(* Logix 5000 project; controller CipDriveFaultCodes vendor 1 type 14 code 156 rev 32.11; software revision 32.02 *)

TASK MainTask (continuous, watchdog 500 ms) : MainProgram

MODULES
   Local : vendor 1 type 14 code 156 (Compact 0, rev 32.11)
      Drive_1 : vendor 1 type 37 code 46 (Ethernet 192.168.1.26, rev 7.8, MotionDiagnostics RPI 1 ms)
END_MODULES

VAR_GLOBAL   (* controller tags *)
   A1_CIPAxisFaultsLSW : DINT;
   A1_CIPAxisFaultsMSW : DINT := 45;
   A1_CIPAxisFaultsRA_LSW : DINT;
   A1_CIPAxisFaultsRA_MSW : DINT;
   A1_CIPInitializationFaults : DINT;
   A1_CIPStartInhibits : INT;
   A1_CIPStartInhibitsRA : INT;
   A1_ModuleAlarmBits : DINT;
   A1_ModuleFaultBits : DINT;
   Axis_1 : AXIS_CIP_DRIVE;
   Drive_CommConnectionOK : BOOL := 1;
   DriveConnectionStatus : DINT := 16#0000_4000;
   ErrorCode : DINT[10] := ([1] := 8192);
   MotionGrop : MOTION_GROUP;
   TempCipAxisFaultsRA : DINT[2];
END_VAR

PROGRAM MainProgram   (* main routine MainRoutine *)

ROUTINE MainRoutine   (* ladder *)
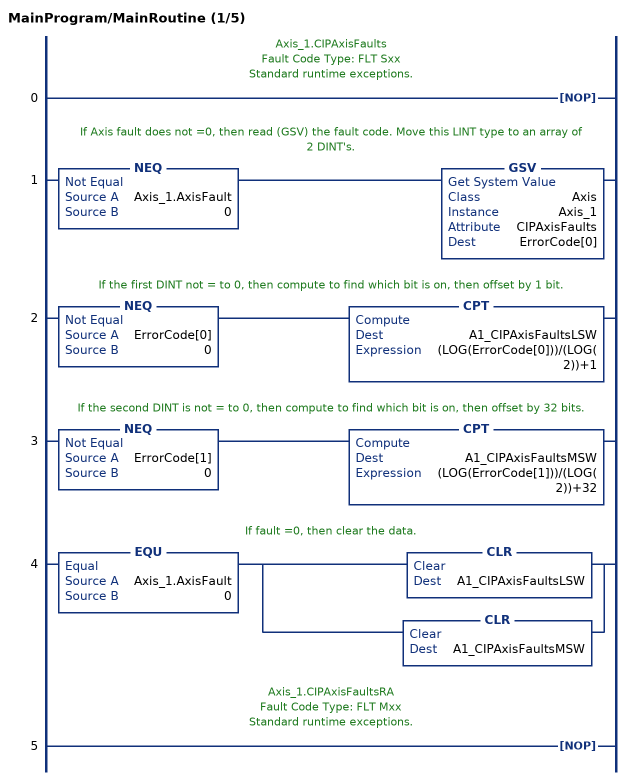
   // Axis_1.CIPAxisFaults
   // Fault Code Type: FLT Sxx
   // Standard runtime exceptions.
   0: NOP();
   // If Axis fault does not =0, then read (GSV) the fault code. Move this LINT type to an array of 2 DINT's.
   1: NEQ(Axis_1.AxisFault,0)GSV(Axis,Axis_1,CIPAxisFaults,ErrorCode[0]);
   // If the first DINT not = to 0, then compute to find which bit is on, then offset by 1 bit.
   2: NEQ(ErrorCode[0],0)CPT(A1_CIPAxisFaultsLSW,(LOG(ErrorCode[0]))/(LOG(2))+1);
   // If the second DINT is not = to 0, then compute to find which bit is on, then offset by 32 bits.
   3: NEQ(ErrorCode[1],0)CPT(A1_CIPAxisFaultsMSW,(LOG(ErrorCode[1]))/(LOG(2))+32);
   // If fault =0, then clear the data.
   4: EQU(Axis_1.AxisFault,0)[CLR(A1_CIPAxisFaultsLSW) ,CLR(A1_CIPAxisFaultsMSW) ];
   // Axis_1.CIPAxisFaultsRA
   // Fault Code Type: FLT Mxx
   // Standard runtime exceptions.
   5: NOP();
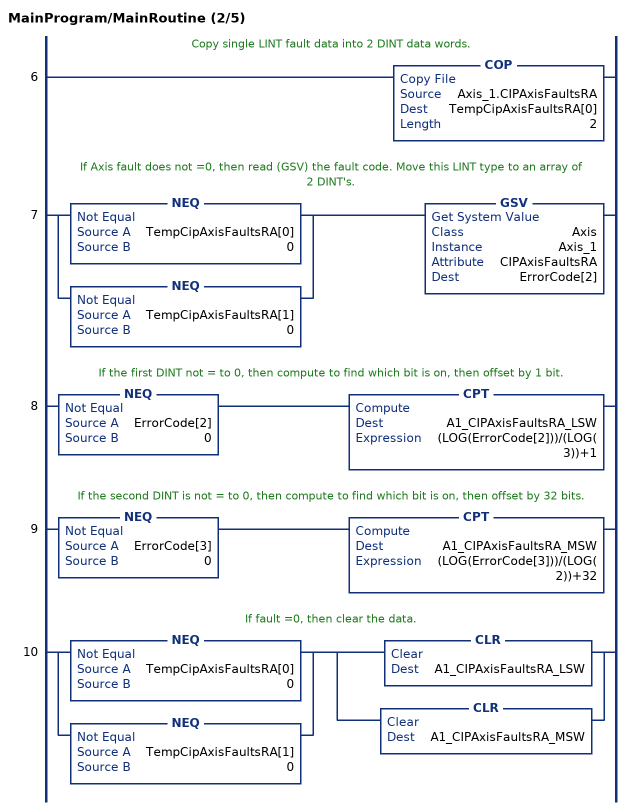
   // Copy single LINT fault data into 2 DINT data words.
   6: COP(Axis_1.CIPAxisFaultsRA,TempCipAxisFaultsRA[0],2);
   // If Axis fault does not =0, then read (GSV) the fault code. Move this LINT type to an array of 2 DINT's.
   7: [NEQ(TempCipAxisFaultsRA[0],0) ,NEQ(TempCipAxisFaultsRA[1],0) ]GSV(Axis,Axis_1,CIPAxisFaultsRA,ErrorCode[2]);
   // If the first DINT not = to 0, then compute to find which bit is on, then offset by 1 bit.
   8: NEQ(ErrorCode[2],0)CPT(A1_CIPAxisFaultsRA_LSW,(LOG(ErrorCode[2]))/(LOG(3))+1);
   // If the second DINT is not = to 0, then compute to find which bit is on, then offset by 32 bits.
   9: NEQ(ErrorCode[3],0)CPT(A1_CIPAxisFaultsRA_MSW,(LOG(ErrorCode[3]))/(LOG(2))+32);
   // If fault =0, then clear the data.
   10: [NEQ(TempCipAxisFaultsRA[0],0) ,NEQ(TempCipAxisFaultsRA[1],0) ][CLR(A1_CIPAxisFaultsRA_LSW) ,CLR(A1_CIPAxisFaultsRA_MSW) ];
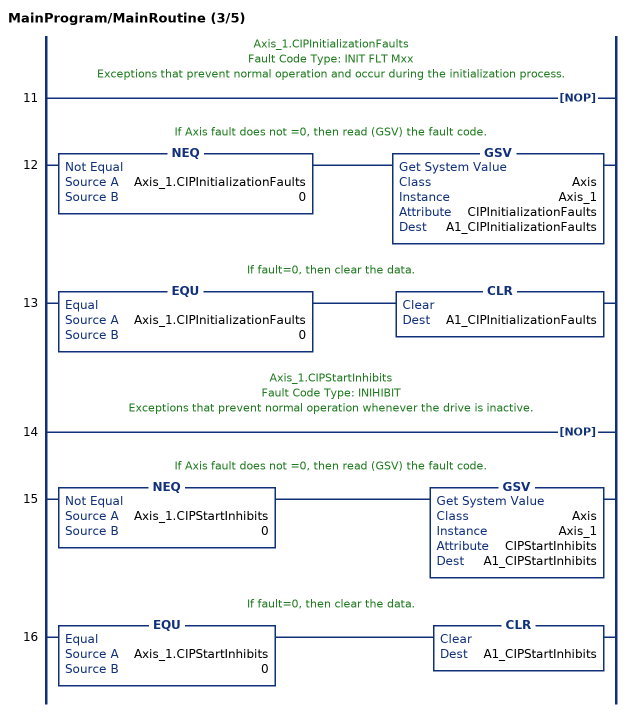
   // Axis_1.CIPInitializationFaults
   // Fault Code Type: INIT FLT Mxx
   // Exceptions that prevent normal operation and occur during the initialization process.
   11: NOP();
   // If Axis fault does not =0, then read (GSV) the fault code.
   12: NEQ(Axis_1.CIPInitializationFaults,0)GSV(Axis,Axis_1,CIPInitializationFaults,A1_CIPInitializationFaults);
   // If fault=0, then clear the data.
   13: EQU(Axis_1.CIPInitializationFaults,0)CLR(A1_CIPInitializationFaults);
   // Axis_1.CIPStartInhibits
   // Fault Code Type: INIHIBIT
   // Exceptions that prevent normal operation whenever the drive is inactive.
   14: NOP();
   // If Axis fault does not =0, then read (GSV) the fault code.
   15: NEQ(Axis_1.CIPStartInhibits,0)GSV(Axis,Axis_1,CIPStartInhibits,A1_CIPStartInhibits);
   // If fault=0, then clear the data.
   16: EQU(Axis_1.CIPStartInhibits,0)CLR(A1_CIPStartInhibits);
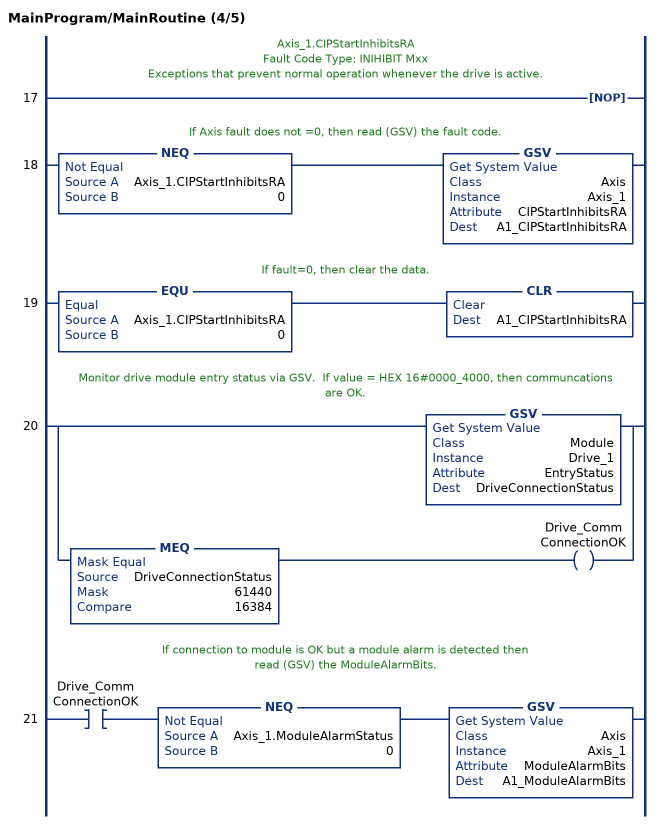
   // Axis_1.CIPStartInhibitsRA
   // Fault Code Type: INIHIBIT Mxx
   // Exceptions that prevent normal operation whenever the drive is active.
   17: NOP();
   // If Axis fault does not =0, then read (GSV) the fault code.
   18: NEQ(Axis_1.CIPStartInhibitsRA,0)GSV(Axis,Axis_1,CIPStartInhibitsRA,A1_CIPStartInhibitsRA);
   // If fault=0, then clear the data.
   19: EQU(Axis_1.CIPStartInhibitsRA,0)CLR(A1_CIPStartInhibitsRA);
   // Monitor drive module entry status via GSV.  If value = HEX 16#0000_4000, then communcations are OK.
   20: [GSV(Module,Drive_1,EntryStatus,DriveConnectionStatus) ,MEQ(DriveConnectionStatus,61440,16384) OTE(Drive_CommConnectionOK) ];
   // If connection to module is OK but a module alarm is detected then
   // read (GSV) the ModuleAlarmBits.
   21: XIC(Drive_CommConnectionOK)NEQ(Axis_1.ModuleAlarmStatus,0)GSV(Axis,Axis_1,ModuleAlarmBits,A1_ModuleAlarmBits);
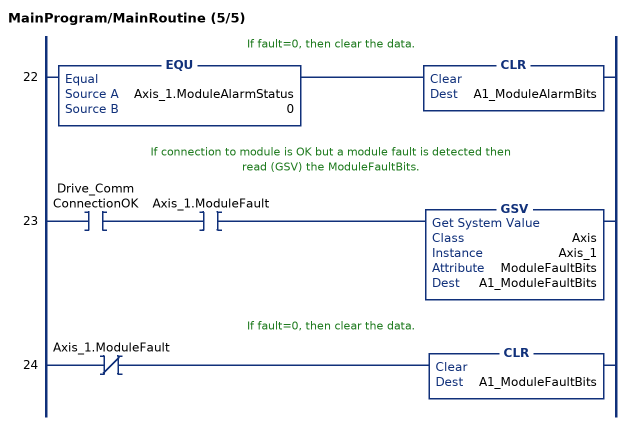
   // If fault=0, then clear the data.
   22: EQU(Axis_1.ModuleAlarmStatus,0)CLR(A1_ModuleAlarmBits);
   // If connection to module is OK but a module fault is detected then
   // read (GSV) the ModuleFaultBits.
   23: XIC(Drive_CommConnectionOK)XIC(Axis_1.ModuleFault)GSV(Axis,Axis_1,ModuleFaultBits,A1_ModuleFaultBits);
   // If fault=0, then clear the data.
   24: XIO(Axis_1.ModuleFault)CLR(A1_ModuleFaultBits);
END_ROUTINE
END_PROGRAM
